// TIA Portal project "Drehstrommotor Funktion 1" (V13)

(* hardware
DEVICE "S7300/ET200M-Station_1"  S7-300 station
   slot 0: "Profilschiene_0"  Rail  6ES7 390-1***0-0AA0
   slot 1: "PS 307 5A_1"  PS 307 5A  6ES7 307-1EA00-0AA0
   slot 2: "SIMATIC S7-300"  CPU 314C-2 PN/DP  6ES7 314-6EH04-0AB0  V3.3
      slot 2: "PROFINET-Schnittstelle_1"  PN-IO
         slot 1: "Port_1"  Port
         slot 2: "Port_2"  Port
      slot 5: "DI 24/DO 16_1"  DI24/DO16
      slot 6: "AI 5/AO 2_1"  AI5/AO2
      slot 7: "Zählen_1"  Counter
      slot 8: "Positionieren_1"  Positioning
   slot 4: "CP 343-2_1"  CP 343-2  6GK7 343-2AH01-0XA0  V3.1
*)

// ===== PLC "SIMATIC S7-300"  CPU 314C-2 PN/DP =====

VAR_GLOBAL   // PLC tag table "Standard-Variablentabelle"
   "S0" AT %I124.0 : Bool;   // Stop I (NC)
   "S1" AT %I124.1 : Bool;   // Start I
   "S3" AT %I124.3 : Bool;   // Stopp II (NC)
   "S4" AT %I124.4 : Bool;   // Start II
   "F2 (S5)" AT %I124.5 : Bool;   // Motorschutzrelasi F2 (NC)
   "Q1" AT %Q124.0 : Bool;   // Leitstunsschütz
   "P1" AT %Q124.7 : Bool;   // Meldelampe
   "MB10" AT %MB10 : Byte;   // Merkerkbyte 10
   "MB20" AT %MB20 : Byte;   // Merkerbyte 20
   "Start Step 1" AT %M20.1 : Bool;   // Starten des Programmes
   "Step 1" AT %M10.1 : Bool;   // Step 1
   "Step 2" AT %M10.2 : Bool;   // Step 2
   "step 0" AT %M10.0 : Bool;   // Step 0
   "0.8S-Takt" AT %M100.4 : Bool;   // 0.8S-Takt
END_VAR

FUNCTION "Grafcet" : Void   // FC1, FBD
{ S7_Optimized_Access := 'FALSE' }
VERSION : 0.1
BEGIN

REGION Network 1: Step 0
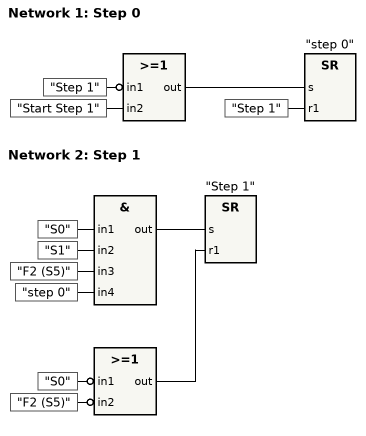
   IF NOT "Step 1" OR "Start Step 1" THEN
       "step 0" := TRUE;   // SR flip-flop
   END_IF;
   IF "Step 1" THEN "step 0" := FALSE; END_IF;
END_REGION

REGION Network 2: Step 1
   IF "S0" AND "S1" AND "F2 (S5)" AND "step 0" THEN
       "Step 1" := TRUE;   // SR flip-flop
   END_IF;
   IF NOT "S0" OR NOT "F2 (S5)" THEN "Step 1" := FALSE; END_IF;
END_REGION
END_FUNCTION

FUNCTION "Actions" : Void   // FC2, FBD
{ S7_Optimized_Access := 'FALSE' }
VERSION : 0.1
BEGIN

REGION Network 1: Motor 1
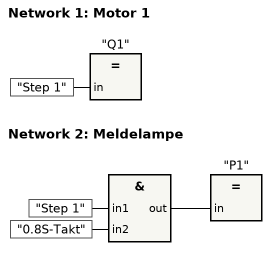
   "Q1" := "Step 1";
END_REGION

REGION Network 2: Meldelampe
   "P1" := "Step 1" AND "0.8S-Takt";
END_REGION
END_FUNCTION

ORGANIZATION_BLOCK "Main"   // OB1, FBD
TITLE = "Main Program Sweep (Cycle)"
{ S7_Optimized_Access := 'FALSE' }
VERSION : 0.1
BEGIN

REGION Network 1
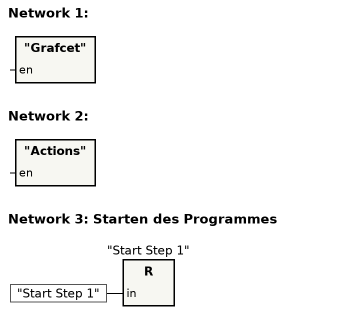
   "Grafcet"();
END_REGION

REGION Network 2
   "Actions"();
END_REGION

REGION Network 3: Starten des Programmes
   IF "Start Step 1" THEN "Start Step 1" := FALSE; END_IF;
END_REGION
END_ORGANIZATION_BLOCK

ORGANIZATION_BLOCK "COMPLETE RESTART"   // OB100, FBD
TITLE = "Complete Restart"
{ S7_Optimized_Access := 'FALSE' }
VERSION : 0.1
BEGIN

REGION Network 1
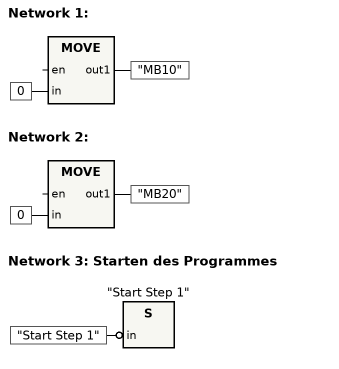
   "MB10" := 0;
END_REGION

REGION Network 2
   "MB20" := 0;
END_REGION

REGION Network 3: Starten des Programmes
   IF NOT "Start Step 1" THEN "Start Step 1" := TRUE; END_IF;
END_REGION
END_ORGANIZATION_BLOCK